{attribute 'GeneratedUsingTerminal: ELM9410-0000-0016'}
{attribute addProperty BoxType "ELM9410-0000-0016"}
{attribute addProperty Id "ValueAT %I*INT2"}
{attribute addProperty CRC "2162654570"}
{attribute addProperty Size "2"}
TYPE MMS_Acceleration_Z_Axis_80E77D6A EXTENDS InputBase_8311D824 :
STRUCT
	{attribute addProperty Name "Value"}
	Value AT %I* : INT;
END_STRUCT
END_TYPE

(* stored: Version 1.2.0.0, ProductVersion 3.1.4024.9
   DUT MMS_Acceleration_Z_Axis_80E77D6A: Id {838af423-c4a8-407b-b0f4-b2f0f4ae455e} *)
